// TIA Portal project "thuc_hanh_1" (V14)

(* hardware
DEVICE "S7-1200 station_1"  S7-1200 Station
   slot 0: "Rack_0"  S7-1200 Rack  Rack  V1.0
   slot 1: "PLC_1"  CPU 1214C DC/DC/DC  6ES7 214-1AG40-0XB0  V4.2
*)

// ===== PLC "PLC_1"  CPU 1214C DC/DC/DC =====

VAR_GLOBAL   // PLC tag table "Default tag table"
   "Tag_1" AT %I0.0 : Bool;
   "xanh" AT %Q0.0 : Bool;
   "Start" AT %I0.3 : Bool;
   "Tag_4" AT %M0.0 : Bool;
   "đỏ" AT %Q0.2 : Bool;
   "Tag_6" AT %I0.1 : Bool;
   "Tag_7" AT %M0.2 : Bool;
   "vàng" AT %Q0.1 : Bool;
   "Tag_9" AT %Q0.3 : Bool;
   "Stop" AT %I0.2 : Bool;
   "Tag_11" AT %Q0.4 : Bool;
   "Tag_12" AT %M0.1 : Bool;
   "Tag_2" AT %M10.0 : Bool;
   "Tag_3" AT %M10.1 : Bool;
   "Tag_5" AT %M10.2 : Bool;
   "Tag_8" AT %M10.3 : Bool;
   "ST1_" AT %M0.3 : Bool;
   "Start_" AT %M0.4 : Bool;
   "T1_" AT %M0.5 : Bool;
   "T2_" AT %M0.6 : Bool;
   "A1_" AT %M0.7 : Bool;
   "reset_" AT %M1.0 : Bool;
   "ST2_" AT %M1.1 : Bool;
   "ST4_" AT %M1.2 : Bool;
   "ST3_" AT %M1.3 : Bool;
   "ST5_" AT %M1.4 : Bool;
   "ST6_" AT %M1.5 : Bool;
   "A2_" AT %M1.6 : Bool;
   "A3_" AT %M1.7 : Bool;
   "A4_" AT %M2.0 : Bool;
   "A5_" AT %M2.1 : Bool;
   "A6_" AT %M2.2 : Bool;
   "A7_" AT %M2.3 : Bool;
   "A8_" AT %M2.4 : Bool;
   "A9_" AT %M2.5 : Bool;
   "A10_" AT %M2.6 : Bool;
   "ST1X_" AT %M2.7 : Bool;
   "ST2X_" AT %M3.0 : Bool;
   "ST3X_" AT %M3.1 : Bool;
   "ST4X_" AT %M3.2 : Bool;
   "ST5X_" AT %M3.3 : Bool;
   "ST6X_" AT %M3.4 : Bool;
   "den_mc" AT %M3.5 : Bool;
   "Team1_xanh" AT %M3.6 : Bool;
   "Team1_do" AT %M3.7 : Bool;
   "Team2_xanh" AT %M4.0 : Bool;
   "Team2_do" AT %M4.1 : Bool;
   "but1" AT %M4.2 : Bool;
   "but2" AT %M4.3 : Bool;
   "but_start" AT %M4.4 : Bool;
   "but_reset" AT %M4.5 : Bool;
   "re" AT %M4.6 : Bool;
END_VAR

ORGANIZATION_BLOCK "Main"   // OB1, LAD, ProgramCycle
TITLE = "Main Program Sweep (Cycle)"
{ S7_Optimized_Access := 'TRUE' }
VERSION : 0.1
   VAR_INPUT
      Initial_Call : Bool;   // Initial call of this OB
      Remanence : Bool;   // =True, if remanent data are available
   END_VAR
BEGIN

REGION Network 1
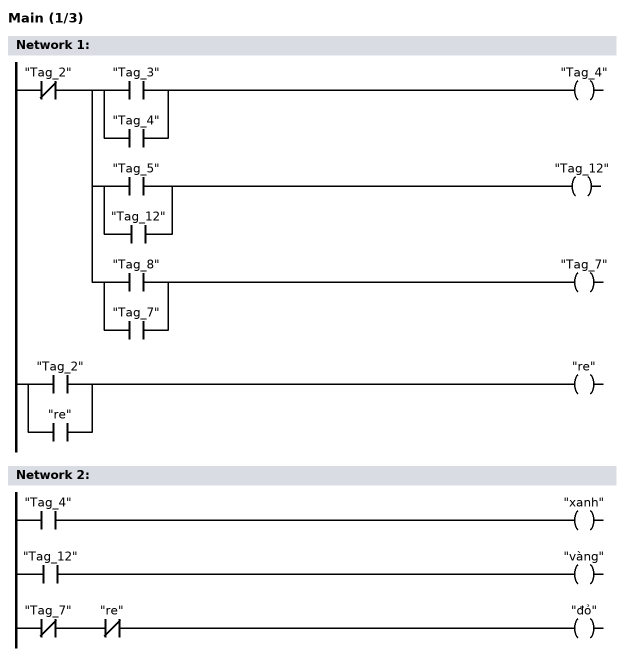
   RUNG wire#powerrail
      I_Contact( "Tag_2" )
      wire#w1
      Contact( "Tag_3" )
      wire#w2
      Coil( "Tag_4" )
   END_RUNG
   RUNG wire#w1
      Contact( "Tag_4" )
   END_RUNG wire#w2
   RUNG wire#w1
      Contact( "Tag_5" )
      wire#w3
      Coil( "Tag_12" )
   END_RUNG
   RUNG wire#w1
      Contact( "Tag_12" )
   END_RUNG wire#w3
   RUNG wire#w1
      Contact( "Tag_8" )
      wire#w4
      Coil( "Tag_7" )
   END_RUNG
   RUNG wire#w1
      Contact( "Tag_7" )
   END_RUNG wire#w4
   RUNG wire#powerrail
      Contact( "Tag_2" )
      wire#w5
      Coil( "re" )
   END_RUNG
   RUNG wire#powerrail
      Contact( "re" )
   END_RUNG wire#w5
   // the same network as SCL:
   "Tag_4" := NOT "Tag_2" AND ("Tag_3" OR "Tag_4");
   "Tag_12" := NOT "Tag_2" AND ("Tag_5" OR "Tag_12");
   "Tag_7" := NOT "Tag_2" AND ("Tag_8" OR "Tag_7");
   "re" := "Tag_2" OR "re";
END_REGION

REGION Network 2
   RUNG wire#powerrail
      Contact( "Tag_4" )
      Coil( "xanh" )
   END_RUNG
   RUNG wire#powerrail
      Contact( "Tag_12" )
      Coil( "vàng" )
   END_RUNG
   RUNG wire#powerrail
      I_Contact( "Tag_7" )
      I_Contact( "re" )
      Coil( "đỏ" )
   END_RUNG
   // the same network as SCL:
   "xanh" := "Tag_4";
   "vàng" := "Tag_12";
   "đỏ" := NOT "Tag_7" AND NOT "re";
END_REGION

REGION Network 3
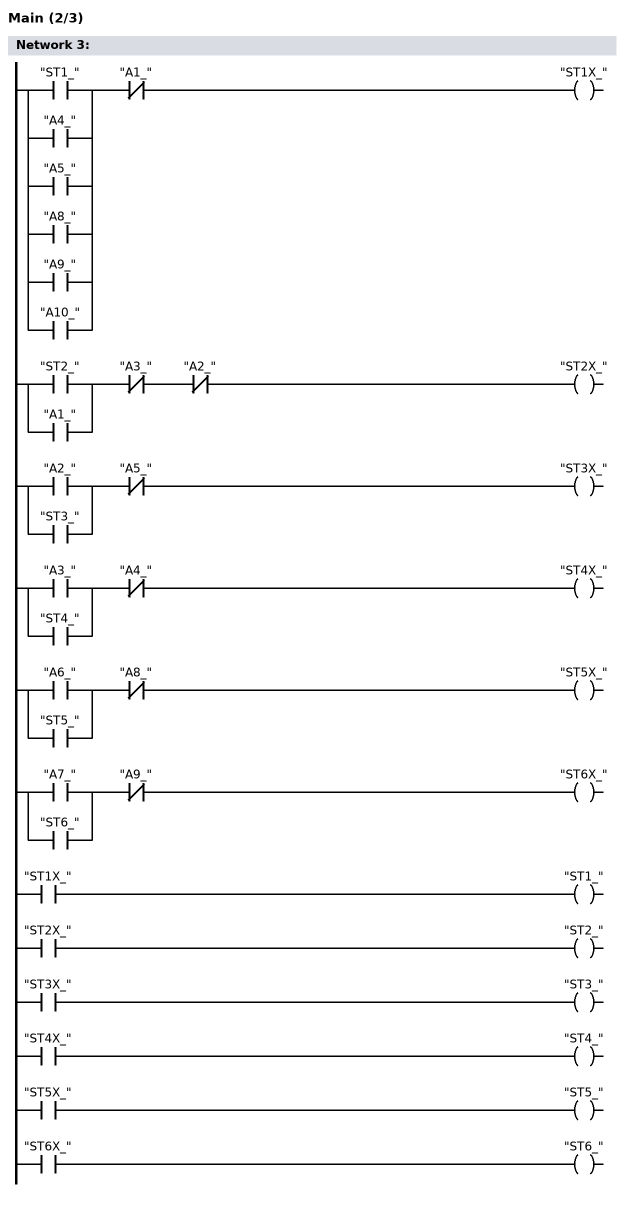
   RUNG wire#powerrail
      Contact( "ST1_" )
      wire#w1
      I_Contact( "A1_" )
      Coil( "ST1X_" )
   END_RUNG
   RUNG wire#powerrail
      Contact( "A4_" )
   END_RUNG wire#w1
   RUNG wire#powerrail
      Contact( "A5_" )
   END_RUNG wire#w1
   RUNG wire#powerrail
      Contact( "A8_" )
   END_RUNG wire#w1
   RUNG wire#powerrail
      Contact( "A9_" )
   END_RUNG wire#w1
   RUNG wire#powerrail
      Contact( "A10_" )
   END_RUNG wire#w1
   RUNG wire#powerrail
      Contact( "ST2_" )
      wire#w2
      I_Contact( "A3_" )
      I_Contact( "A2_" )
      Coil( "ST2X_" )
   END_RUNG
   RUNG wire#powerrail
      Contact( "A1_" )
   END_RUNG wire#w2
   RUNG wire#powerrail
      Contact( "A2_" )
      wire#w3
      I_Contact( "A5_" )
      Coil( "ST3X_" )
   END_RUNG
   RUNG wire#powerrail
      Contact( "ST3_" )
   END_RUNG wire#w3
   RUNG wire#powerrail
      Contact( "A3_" )
      wire#w4
      I_Contact( "A4_" )
      Coil( "ST4X_" )
   END_RUNG
   RUNG wire#powerrail
      Contact( "ST4_" )
   END_RUNG wire#w4
   RUNG wire#powerrail
      Contact( "A6_" )
      wire#w5
      I_Contact( "A8_" )
      Coil( "ST5X_" )
   END_RUNG
   RUNG wire#powerrail
      Contact( "ST5_" )
   END_RUNG wire#w5
   RUNG wire#powerrail
      Contact( "A7_" )
      wire#w6
      I_Contact( "A9_" )
      Coil( "ST6X_" )
   END_RUNG
   RUNG wire#powerrail
      Contact( "ST6_" )
   END_RUNG wire#w6
   RUNG wire#powerrail
      Contact( "ST1X_" )
      Coil( "ST1_" )
   END_RUNG
   RUNG wire#powerrail
      Contact( "ST2X_" )
      Coil( "ST2_" )
   END_RUNG
   RUNG wire#powerrail
      Contact( "ST3X_" )
      Coil( "ST3_" )
   END_RUNG
   RUNG wire#powerrail
      Contact( "ST4X_" )
      Coil( "ST4_" )
   END_RUNG
   RUNG wire#powerrail
      Contact( "ST5X_" )
      Coil( "ST5_" )
   END_RUNG
   RUNG wire#powerrail
      Contact( "ST6X_" )
      Coil( "ST6_" )
   END_RUNG
   // the same network as SCL:
   "ST1X_" := ("ST1_" OR "A4_" OR "A5_" OR "A8_" OR "A9_" OR "A10_") AND NOT "A1_";
   "ST2X_" := ("ST2_" OR "A1_") AND NOT "A3_" AND NOT "A2_";
   "ST3X_" := ("A2_" OR "ST3_") AND NOT "A5_";
   "ST4X_" := ("A3_" OR "ST4_") AND NOT "A4_";
   "ST5X_" := ("A6_" OR "ST5_") AND NOT "A8_";
   "ST6X_" := ("A7_" OR "ST6_") AND NOT "A9_";
   "ST1_" := "ST1X_";
   "ST2_" := "ST2X_";
   "ST3_" := "ST3X_";
   "ST4_" := "ST4X_";
   "ST5_" := "ST5X_";
   "ST6_" := "ST6X_";
END_REGION

REGION Network 4
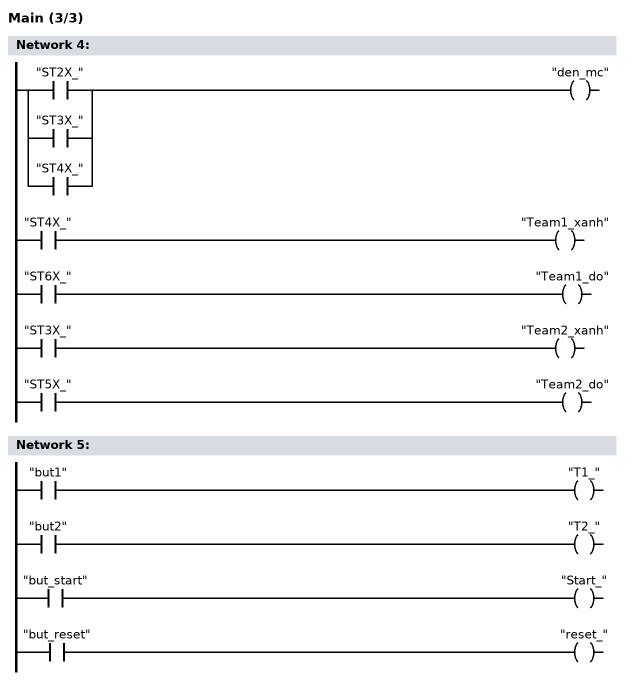
   RUNG wire#powerrail
      Contact( "ST2X_" )
      wire#w1
      Coil( "den_mc" )
   END_RUNG
   RUNG wire#powerrail
      Contact( "ST3X_" )
   END_RUNG wire#w1
   RUNG wire#powerrail
      Contact( "ST4X_" )
   END_RUNG wire#w1
   RUNG wire#powerrail
      Contact( "ST4X_" )
      Coil( "Team1_xanh" )
   END_RUNG
   RUNG wire#powerrail
      Contact( "ST6X_" )
      Coil( "Team1_do" )
   END_RUNG
   RUNG wire#powerrail
      Contact( "ST3X_" )
      Coil( "Team2_xanh" )
   END_RUNG
   RUNG wire#powerrail
      Contact( "ST5X_" )
      Coil( "Team2_do" )
   END_RUNG
   // the same network as SCL:
   "den_mc" := "ST2X_" OR "ST3X_" OR "ST4X_";
   "Team1_xanh" := "ST4X_";
   "Team1_do" := "ST6X_";
   "Team2_xanh" := "ST3X_";
   "Team2_do" := "ST5X_";
END_REGION

REGION Network 5
   RUNG wire#powerrail
      Contact( "but1" )
      Coil( "T1_" )
   END_RUNG
   RUNG wire#powerrail
      Contact( "but2" )
      Coil( "T2_" )
   END_RUNG
   RUNG wire#powerrail
      Contact( "but_start" )
      Coil( "Start_" )
   END_RUNG
   RUNG wire#powerrail
      Contact( "but_reset" )
      Coil( "reset_" )
   END_RUNG
   // the same network as SCL:
   "T1_" := "but1";
   "T2_" := "but2";
   "Start_" := "but_start";
   "reset_" := "but_reset";
END_REGION
END_ORGANIZATION_BLOCK